FUNCTION_BLOCK FB_DoubleCoilCylinder2 EXTENDS FB_SingleCoilCylinder
VAR_INPUT
END_VAR
VAR_OUTPUT
END_VAR
VAR
	(* Coils *)
	poHomeValve	: FB_DigitalOutput;	(* Home position valve function block *)
END_VAR

IF bFirstCycle THEN
	poActiveValve.MR_FirstCycle( sName := CONCAT(sName,':Home_Valve'),sModuleType := ref_poHomeValve.ModuleType, sPortID := ref_poHomeValve.PortID);	
END_IF

SUPER^();

bPositionHold := poActiveValve.Out OR poHomeValve.Out;

poHomeValve();

METHOD MR_GoActive : BOOL
IF eCylinderState = CYLINDER_IDLE AND NOT poActiveValve.Out THEN
	bBusy := TRUE;
	bGoActive := TRUE;
	MR_GoActive := FALSE;
	eCylinderState := CYLINDER_GO_ACTIVE;
	eCylinderGoActiveState := CYLINDER_MOVE_START_TRACKING;
	fbMachineLogger.MR_AddLogs(CONCAT(sName,' : active position requested'));	
	
	
ELSIF eCylinderState = CYLINDER_GO_ACTIVE_DONE THEN
	bGoActive := FALSE;
	MR_GoActive := TRUE;
	fbMachineLogger.MR_AddLogs(CONCAT(sName,' : active position done'));		
	
END_IF
END_METHOD

METHOD MR_GoHome : BOOL
IF eCylinderState = CYLINDER_IDLE AND NOT poHomeValve.Out THEN
	bBusy := TRUE;
	bGoHome := TRUE;
	MR_GoHome := FALSE;
	eCylinderState := CYLINDER_GO_HOME;
	eCylinderGoHomeState := CYLINDER_MOVE_START_TRACKING;
	fbMachineLogger.MR_AddLogs(CONCAT(sName,' : home position requested'));	
	
ELSIF eCylinderState = CYLINDER_GO_HOME_DONE THEN
	bGoHome := FALSE;
	MR_GoHome := TRUE;
	fbMachineLogger.MR_AddLogs(CONCAT(sName,' : home position done'));	
	
END_IF
END_METHOD

METHOD PROTECTED MS_GoActive
VAR_INPUT
END_VAR
poHomeValve.Out := FALSE;
SUPER^.MS_GoActive();
END_METHOD

METHOD PROTECTED MS_GoHome
VAR_INPUT
END_VAR
poHomeValve.Out := TRUE;
SUPER^.MS_GoHome();
END_METHOD

METHOD PROTECTED MS_Release
VAR_INPUT
END_VAR
poHomeValve.Out := FALSE;
SUPER^.MS_Release();
END_METHOD

METHOD PROTECTED MS_Reset
VAR_INPUT
END_VAR
poHomeValve.Out := FALSE;

SUPER^.MS_Reset();
END_METHOD

METHOD PROTECTED MS_Uninitialized
poHomeValve.Out := FALSE;
SUPER^.MS_Uninitialized();
END_METHOD

PROPERTY ref_poHomeValve : REFERENCE TO FB_DigitalOutput
GET
ref_poHomeValve REF= poHomeValve;
END_GET
END_PROPERTY

END_FUNCTION_BLOCK

(* stored: Version 1.1.0.1, ProductVersion 3.1.4024.9
   POU FB_DoubleCoilCylinder2: Id {6394a067-a605-4841-94b9-6e88d67a6233}, SpecialFunc None
   Folder Properties: Id {2ff649ee-b3b2-45fd-a5ba-7f938608f4ae}
   Folder Status: Id {a0cebb56-33c1-45b7-a76e-5a06e8c01b2e}
   Folder Requests: Id {1026cab6-2aea-49ef-aa8d-59dd3baa5fc3}
   Folder State Machine: Id {3c5d73bb-f649-4315-aaa5-acf0e3766f10}
   Method MR_GoActive: Id {3d8f36f0-62ce-4576-9ece-6139bbaf9818}
   Method MR_GoHome: Id {f652d8ad-fbda-44d7-a81b-d925edae764e}
   Method MS_GoActive: Id {8ee272ed-250f-441e-8f41-26907d0b619d}
   Method MS_GoHome: Id {79f64506-08d6-42e6-873b-72c162ab1ade}
   Method MS_Release: Id {24956562-7df7-4811-82e2-ef448db60d14}
   Method MS_Reset: Id {aece39ae-c62c-45b8-8902-3385fe888dd3}
   Method MS_Uninitialized: Id {47355d1b-3e3f-45a0-8e4d-f18a081d452a}
   Property ref_poHomeValve: Id {c8d0dca1-d468-413d-9174-2fa008d052f3}
   Get Get: Id {4aef4ded-2005-451c-9096-fe6f77f38fc0} *)
